{attribute 'GeneratedUsingTerminal: EL9520-0000-0016'}
{attribute addProperty BoxType "EL9520-0000-0016"}
{attribute addProperty Id "EtcSlaveTerminalBasePowerOKAT %I*PowerOK_CEB2FD121WcStateAT %I*WcState_9091E0EB2InfoDataAT %I*InfoData_6F19DB2B2"}
{attribute addProperty CRC "851740164"}
{attribute addProperty Size "5"}
TYPE EL9520_32C48604 EXTENDS EtcSlaveTerminalBase :
STRUCT
	{attribute addProperty Name "PowerOK"}
	PowerOK : PowerOK_CEB2FD12;
	{attribute addProperty Name "WcState"}
	WcState : WcState_9091E0EB;
	{attribute addProperty Name "InfoData"}
	InfoData : InfoData_6F19DB2B;
END_STRUCT
END_TYPE

(* stored: Version 1.2.0.0, ProductVersion 3.1.4024.9
   DUT EL9520_32C48604: Id {18c8fe6b-ea75-481c-bc52-1802bfbb2210} *)
